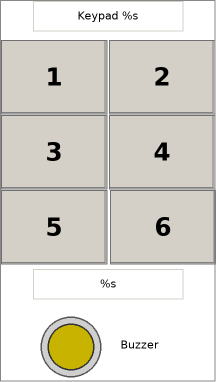
VISUALIZATION Keypad  // 216x382
VAR_IN_OUT
	stKeypadVirtual	: ST_AlarmKeypadVirtual;
	stKeypad		: ST_AlarmKeypadHMI;
END_VAR
    Button (1,40 106x74), "1", colour toggle: stKeypad.bLed1
        tap stKeypadVirtual.bButton1
    Button (109,40 106x74), "2", colour toggle: stKeypad.bLed2
        tap stKeypadVirtual.bButton2
    Button (1,115 106x74), "3", colour toggle: stKeypad.bLed3
        tap stKeypadVirtual.bButton3
    Button (109,115 106x74), "4", colour toggle: stKeypad.bLed4
        tap stKeypadVirtual.bButton4
    Button (1,190 106x74), "5", colour toggle: stKeypad.bLed5
        tap stKeypadVirtual.bButton5
    Button (110,190 106x74), "6", colour toggle: stKeypad.bLed6
        tap stKeypadVirtual.bButton6
    Lamp1 (36,312 70x70), variable: stKeypad.bBuzzer, style: Lamp-Lamp1-Yellow
    Label (115,330 49x30), "Buzzer"
    Textfield (33,269 150x30), "%s", text variable: stKeypad.sCode
    Textfield (33,1 150x30), "Keypad %s", text variable: stKeypad.sName
END_VISUALIZATION

(* stored: Version 1.1.0.1, ProductVersion 3.1.4024.12
   Visu Keypad: Id {87c32e02-b77a-4f38-9d1c-3c64a5236637} *)
